FUNCTION_BLOCK Robot
VAR_INPUT
	EN				:BOOL;
	iStartPB		:BOOL;
	iEMR_Stop		:BOOL;
END_VAR
VAR_OUTPUT
	ENO				: BOOL;
	RobotHOME		: BOOL;
	RobotBusy		:BOOL;
	RobotDone		:BOOL;
END_VAR
VAR
	MH_Time		:TON;
	StepNo		:INT;
	MHProgramNo	:INT;
	RobotStart	:BOOL;	
END_VAR

IF iEMR_Stop THEN 
StepNo := 0;	
END_IF

CASE StepNo OF
0:   RobotHOME := TRUE;
     RobotBusy := FALSE;
	 MH_Time(IN :=FALSE);
	 RobotDone := FALSE;
    IF iStartPB AND NOT iEMR_Stop THEN
       StepNo := 10;
    END_IF;

10:
    MHProgramNo := 1;
	RobotBusy := TRUE;
	RobotHOME := FALSE;
    StepNo := 20;

20:
	MH_Time(IN := TRUE, PT :=T#5S);
   IF MH_Time.Q THEN
		RobotDone := TRUE; 
		RobotStart := FALSE; 
		RobotBusy := FALSE;
		StepNo := 30;
    END_IF;

30:
    IF RobotDone THEN
       StepNo := 0;
    END_IF;

END_CASE;

END_FUNCTION_BLOCK

(* stored: Version 1.1.0.1, ProductVersion 3.1.4024.16
   POU Robot: Id {07ec3510-0392-4579-9d5c-d04799bdbf20}, SpecialFunc None *)
